FUNCTION_BLOCK setTimers (* Composite Function Block Type *)
  (* Standard: 61499-2 *)
  (* Version 0.2, 2003-12-05, JHC, Rockwell Automation, Renamed from NEWCOMPFB. *)
  (* Version 0.1, 2002-01-08, JHC, Rockwell Automation, Added DLY FB as example. *)
  (* Version 0.0, 2000-05-27, JHC, Rockwell Automation *)
  (* Compiler header: package fb.rt.template; *)
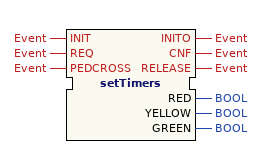
  EVENT_INPUT
    INIT; (* Initialization Request *)
    REQ; (* Normal Execution Request *)
    PEDCROSS;
  END_EVENT
  EVENT_OUTPUT
    INITO; (* Initialization Confirm *)
    CNF; (* Execution Confirmation *)
    RELEASE;
  END_EVENT
  VAR_OUTPUT
    RED : BOOL;
    YELLOW : BOOL;
    GREEN : BOOL;
  END_VAR
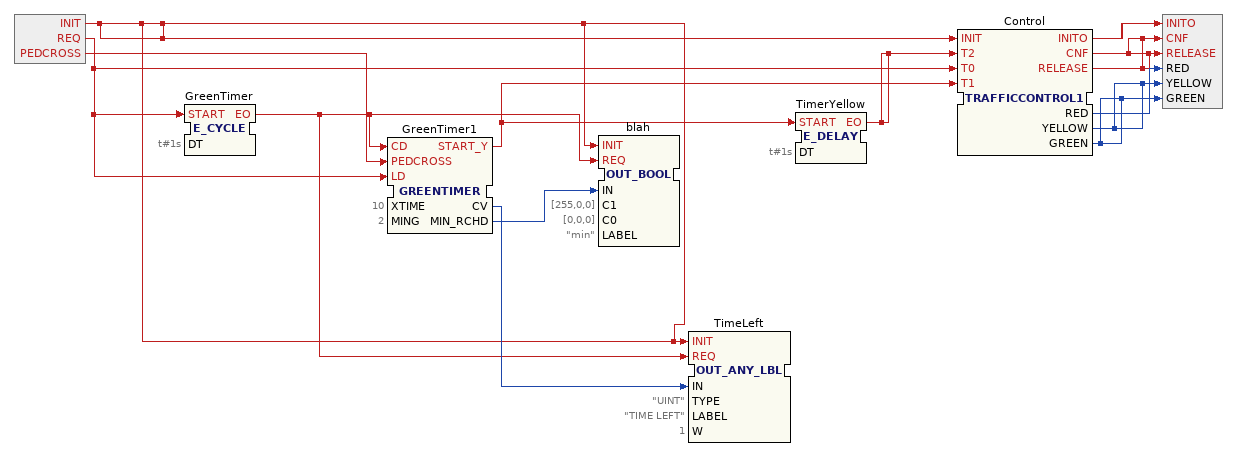
  FBS
    Control : TRAFFICCONTROL1;
    TimerYellow : E_DELAY(DT := t#1s);
    TimeLeft : OUT_ANY_LBL(TYPE := "UINT", LABEL := "TIME LEFT", W := 1);
    GreenTimer : E_CYCLE(DT := t#1s);
    GreenTimer1 : GREENTIMER(XTIME := 10, MING := 2);
    blah : OUT_BOOL(C1 := [255,0,0], C0 := [0,0,0], LABEL := "min");
  END_FBS
  EVENT_CONNECTIONS
    INIT TO Control.INIT;
    TimerYellow.EO TO Control.T2;
    Control.INITO TO INITO;
    Control.CNF TO CNF;
    REQ TO Control.T0;
    Control.RELEASE TO RELEASE;
    INIT TO TimeLeft.INIT;
    REQ TO GreenTimer.START;
    GreenTimer.EO TO TimeLeft.REQ;
    INIT TO Control.INIT;
    TimerYellow.EO TO Control.T2;
    Control.INITO TO INITO;
    Control.CNF TO CNF;
    REQ TO Control.T0;
    Control.RELEASE TO RELEASE;
    INIT TO TimeLeft.INIT;
    REQ TO GreenTimer.START;
    GreenTimer.EO TO TimeLeft.REQ;
    GreenTimer.EO TO GreenTimer1.CD;
    GreenTimer1.START_Y TO Control.T1;
    PEDCROSS TO GreenTimer1.PEDCROSS;
    REQ TO GreenTimer1.LD;
    GreenTimer1.START_Y TO TimerYellow.START;
    INIT TO blah.INIT;
    GreenTimer.EO TO blah.REQ;
  END_CONNECTIONS
  DATA_CONNECTIONS
    Control.RED TO RED;
    Control.YELLOW TO YELLOW;
    Control.GREEN TO GREEN;
    Control.RED TO RED;
    Control.YELLOW TO YELLOW;
    Control.GREEN TO GREEN;
    GreenTimer1.CV TO TimeLeft.IN;
    GreenTimer1.MIN_RCHD TO blah.IN;
  END_CONNECTIONS
END_FUNCTION_BLOCK
